// TIA Portal V20 export
TYPE "LER_typeEmRelationEm_04"
// stored: Access Published, Namespace Unit1
   STRUCT
      commonBit : Array[0..99] of Bool;
      commonInt : Array[0..10] of Int;
      loadingBit : Array[0..99] of Bool;
      attachmentBit : Array[0..99] of Bool;
      fixStageBit : Array[0..99] of Bool;
      loadingInt : Array[0..99] of Int;
      attachmentInt : Array[0..99] of Int;
      fixStageInt : Array[0..99] of Int;
      partData : "LER_typePartData";
      homeCheck : Array[0..31] of Bool;
      homed : Array[0..31] of Bool;
      axis : Array[0..31] of Struct
         interlock : Array[0..99] of Bool;
         inposDone : Array[0..99] of Bool;
         inposDoneBefore : Array[0..99] of Bool;
         inposDoneAfter : Array[0..99] of Bool;
         Moving : Array[0..99] of Bool;
      END_STRUCT;
      cylinder : Array[0..31] of Struct
         inHomePosInterlock : Bool;
         inWorkPosInterlock : Bool;
         inHomePosDone : Bool;
         inWorkPosDone : Bool;
      END_STRUCT;
      digitalSignal : Array[0..31] of Bool;
      loading : Struct
         request : Array[0..31] of Bool;
         ready : Array[0..31] of Bool;
         done : Array[0..31] of Bool;
      END_STRUCT;
      unloading : Struct
         request : Array[0..31] of Bool;
         ready : Array[0..31] of Bool;
         done : Array[0..31] of Bool;
      END_STRUCT;
      clamp : Struct
         request : Array[0..31] of Bool;
         ready : Array[0..31] of Bool;
         done : Array[0..31] of Bool;
      END_STRUCT;
      unclamp : Struct
         request : Array[0..31] of Bool;
         ready : Array[0..31] of Bool;
         done : Array[0..31] of Bool;
      END_STRUCT;
      working : Struct
         ready : Array[0..31] of Bool;
         done : Array[0..31] of Bool;
      END_STRUCT;
      sequence : Array[0..9] of Struct
         job : Array[0..9] of Struct
            locked : Bool;
            active : Bool;
            completed : Bool;
            aborted : Bool;
         END_STRUCT;
      END_STRUCT;
      "r&r" : Struct
         thickness : Struct
            select : Bool;
            workingDone : Bool;
         END_STRUCT;
         vision : Struct
            select : Bool;
            workingDone : Bool;
         END_STRUCT;
         weight : Struct
            select : Bool;
            workingDone : Bool;
         END_STRUCT;
      END_STRUCT;
   END_STRUCT;
END_TYPE
